FUNCTION_BLOCK BaseBlock
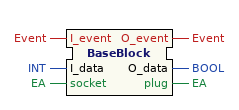
  EVENT_INPUT
    I_event;
  END_EVENT
  EVENT_OUTPUT
    O_event;
  END_EVENT
  VAR_INPUT
    I_data : INT;
  END_VAR
  VAR_OUTPUT
    O_data : BOOL;
  END_VAR
  SOCKETS
    socket : EA;
  END_SOCKETS
  PLUGS
    plug : EA;
  END_PLUGS
  EC_STATES
    START : s -> plug.O_event1;
    Test;
  END_STATES
  ALGORITHM s IN ST:
  VAR_TEMP
    a : INT;
  END_VAR
a := 1;&#38;#10;
  END_ALGORITHM
END_FUNCTION_BLOCK
